{attribute 'qualified_only'}
{attribute 'strict'}
TYPE E_Line :
(
	UnloadElevator := 1,
	UnloadUC,
	Line1,
	Line2,
	Line3
	
);
END_TYPE

(* stored: Version 1.1.0.1, ProductVersion 3.1.4024.3
   DUT E_Line: Id {0426f839-584b-43aa-a08f-2e8733f96801} *)
